PROGRAM MAIN
VAR
	Axis1: AXIS_REF;
	bSTO1 AT %I*: BOOL;
	bSTO2 AT %I*: BOOL;
	fbPower1: MC_POWER;
	bLimFwd1 AT %I*: BOOL;
	bLimBwd1 AT %I*: BOOL;
	Axis2: AXIS_REF;
	fbPower2: MC_POWER;
	bLimFwd2 AT %I*: BOOL;
	bLimBwd2 AT %I*: BOOL;
END_VAR

fbPower1(Axis:=Axis1,
	Enable:=bSTO1 AND bSTO2,
	Enable_Positive:=bLimFwd1,
	Enable_Negative:=bLimBwd1);
fbPower2(Axis:=Axis2,
	Enable:=bSTO1 AND bSTO2,
	Enable_Positive:=bLimFwd2,
	Enable_Negative:=bLimBwd2);

END_PROGRAM

(* stored: Version 1.1.0.1, ProductVersion 3.1.4020.12
   POU MAIN: Id {d369ffcb-6827-470a-b659-0c129921b132}, SpecialFunc None *)
